// TIA Portal V17 export
// export: Created 2025-03-10T13:13:02.1631504Z, ExportSetting WithDefaults, DisplayName Totally Integrated Automation Portal, DisplayVersion V17 Update 8, DisplayName TIA Portal Openness, DisplayVersion V17 Update 8, DisplayName TIA Portal Version Control Interface, DisplayVersion V17, DisplayName SINAMICS Startdrive Advanced, DisplayVersion V17 SP2, DisplayName SINAMICS Startdrive G110M, G120, G120C, G120D, G120P, G115D, DisplayVersion V17 SP2, DisplayName SINAMICS Startdrive G130, G150, S120, S150, SINAMICS MV, S210, DisplayVersion V17 SP2, DisplayName STEP 7 Professional, DisplayVersion V17 Update 8, DisplayName SINUMERIK ONE STEP 7 Toolbox, DisplayVersion V17 Update 12, DisplayName SINUMERIK 840D sl STEP 7 Toolbox, DisplayVersion V17 Update 12, DisplayName STEP 7 Safety, DisplayVersion V17 Update 6, DisplayName WinCC Advanced, DisplayVersion V17 Update 8
DATA_BLOCK "DB22117_MASS_SENSOR_HOPPER_2_UNIT_01"   // DB22117
{ DB_Accessible_From_OPC_UA := 'FALSE' }
VERSION : 0.1
// stored: AutoNumber false, DBAccessibleFromOPCUA false, DBAccessibleFromWebserver true, InstanceOfName FB22105_MASS_SENSOR, InstanceOfType FB
"FB22105_MASS_SENSOR"
   // VAR_INPUT
   //    INPUT_VALUE : Real;
   //    CLEAR_INTERNAL_LOG : Bool;
   //    "SAVE MAX VALUES" : Bool;
   // END_VAR
   // VAR_OUTPUT
   //    OUT_OF_LIMITS_WARNING : Bool;
   //    OUT_OF_LIMITS_ALARM : Bool;
   // END_VAR
   // VAR
   //    OUTPUT : Struct
   //       POWDER_WEIGHT : Real;
   //    END_STRUCT;
   //    INPUT_SETTINGS : Struct
   //       UNIT_NUMBER : DInt := 1;
   //       HOPPER_NUMBER : DInt := 2;
   //    END_STRUCT;
   //    ALARMS_SETTINGS : Struct
   //       LOWER_LIMIT_WARNING : Real;
   //       LOWER_LIMIT_ALARM : Real;
   //       HIGHER_LIMIT_WARNING : Real;
   //       HIGHER_LIMIT_ALARM : Real;
   //       CONFIGURATION_ERROR_ALARM : Bool;
   //    END_STRUCT;
   //    LOG : Struct
   //       DATE_MAX_MASS : Date_And_Time;
   //       VALUE_MAX_MASS : Real;
   //    END_STRUCT;
   // END_VAR
BEGIN
END_DATA_BLOCK
